ABB RobotStudio station: Práctica5_inicio.rspag

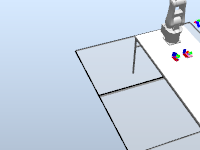
--- station ---
Station Práctica3_inicio (saved by RobotStudio 20.1.9056.2)
Controller Controlador2, task T_ROB1: task frame (RAPID world) sits at (0, 0, 670) mm in the station
Controller Controlador2
  mechanical unit ROB_1: IRB120_3_58__01, 6 joints, base frame (0, 0, 0) mm
Layout (positions relative to the parent item):
  - TVentosa [mechanism] at (-70, 0, 1604) mm
      TCP TVentosa at (0, 0, 51.19) mm
      links: Mi_herramienta
  - LogicGate [smart component, from Components\LogicGate.rslib]
      properties: Operator=NOT; Delay=0
  - LogicGate_2 [smart component, from Components\LogicGate.rslib]
      properties: Operator=AND; Delay=0
  - IRB120_3_58__01 [mechanism, from Robots\IRB120_3_58_G_01.rslib] at (0, 0, 670) mm; joint values [0, 0, -1.5708, 0, 0, 0] (rad or m)
  - table [part, from Libraries\e293a11e-ed86-4237-866f-a9bf8f4bd145table.rslib] at (-246.62, 300, 670) mm, rotated rx 0 ry 0 rz -90 deg
  - Base2 [part]
  - Base1 [part]
  - Detacher [smart component, from Components\Detacher.rslib]
      properties: Child=(none); KeepPosition=true
  - CollisionSensor [smart component, from Components\CollisionSensor.rslib]
      properties: Object1=TVentosa; Object2=(none); NearMiss=0.001; Part1=(none); Part2=(none); CollisionType=0
  - Attacher_2 [smart component, from Components\Attacher.rslib]
      properties: Parent=TVentosa; Flange=0; Child=(none); Mount=false; Offset=[0 0 0]; Orientation=[0 0 0]
  - Source_2 [smart component, from Components\Source.rslib]
      properties: Source=Pieza; Copy=(none); Parent=(none); Position=[0.34 -0.13 0.68]; Orientation=[0 0 0]; Transient=true; PhysicsBehavior=0
  - SimulationEvents_2 [smart component, from Components\SimulationEvents.rslib]
  - Pieza [part] at (340, -130, 700) mm, rotated rx 180 ry 0 rz 180 deg
Attachment: TVentosa is attached to IRB120_3_58__01 / Link6
Attachment: Base2 is attached to Base1
Attachment: Base1 is attached to table
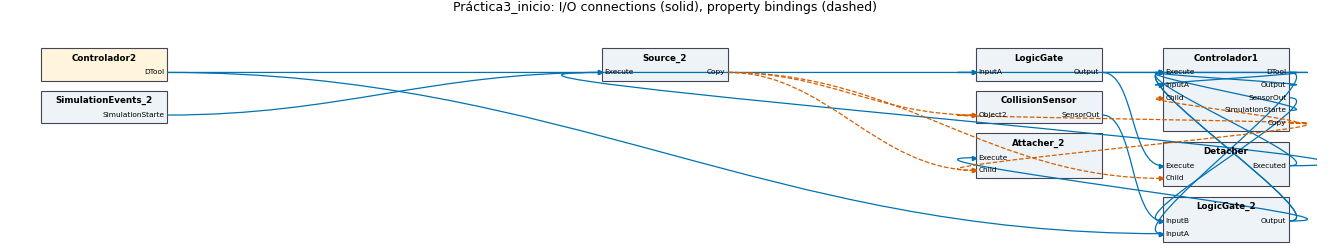
Station logic (signal -> signal, property => property):
  Controlador1.DTool -> Attacher.Execute
  Controlador1.DTool -> LogicGate_2.InputA
  LogicGate_2.Output -> Detacher.Execute
  Controlador1.DTool -> LogicGate.InputA
  LogicGate.Output -> Detacher.Execute
  CollisionSensor.SensorOut -> LogicGate_2.InputB
  Controlador1.DTool -> LogicGate_2.InputA
  LogicGate_2.Output -> Attacher.Execute
  Controlador2.DTool -> LogicGate.InputA
  LogicGate.Output -> Detacher.Execute
  Controlador2.DTool -> LogicGate_2.InputA
  LogicGate_2.Output -> Attacher.Execute
  Detacher.Executed -> Source.Execute
  SimulationEvents.SimulationStarted -> Source.Execute
  CollisionSensor.SensorOut -> LogicGate_2.InputB
  SimulationEvents_2.SimulationStarted -> Source_2.Execute
  Detacher.Executed -> Source_2.Execute
  LogicGate_2.Output -> Attacher_2.Execute
  Source.Copy => Attacher.Child
  Source.Copy => CollisionSensor.Object2
  Source.Copy => Attacher_2.Child
  Source_2.Copy => Attacher_2.Child
  Source_2.Copy => CollisionSensor.Object2
  Source_2.Copy => Detacher.Child

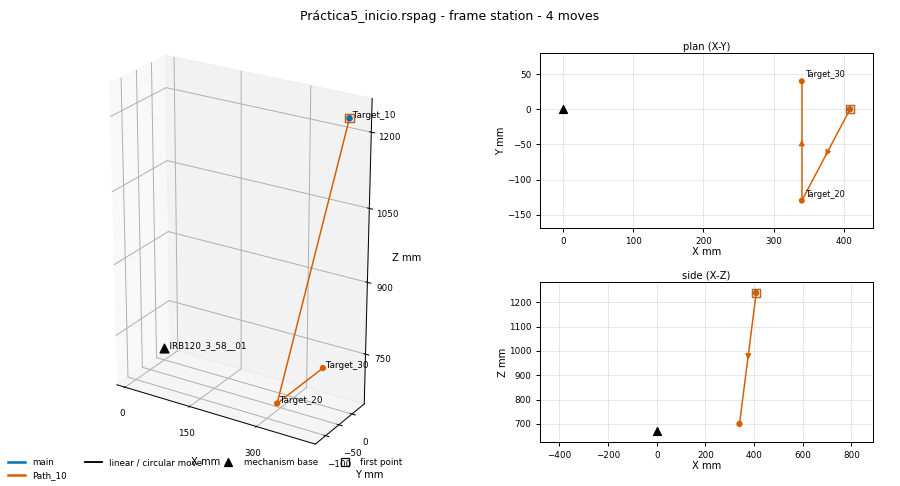
[picture p0: tool path of Práctica5_inicio.rspag in frame station, 4 of 12 moves have a stored position in this frame; points joined in program order, loops and branches not executed]
--- Backups/Controlador2/RAPID/TASK1/PROGMOD/CalibData.mod ---
MODULE CalibData
    PERS tooldata TVentosa:=[TRUE,[[0,0,51.19],[1,0,0,0]],[0.1,[0,0,1],[1,0,0,0],0,0,0]];
    TASK PERS wobjdata WO_Pieza:=[FALSE,TRUE,"",[[300,-150,10],[1,0,0,0]],[[20,10,0],[1,0,0,0]]];
    TASK PERS wobjdata WO_Base2:=[FALSE,TRUE,"",[[300,-150,10],[1,0,0,0]],[[0,150,0],[1,0,0,0]]];
ENDMODULE

--- Backups/Controlador2/RAPID/TASK1/PROGMOD/Module1.mod ---
MODULE Module1
    CONST robtarget Target_10:=[[408.685,0,568.405],[0.5,0,0.866025404,0],[0,0,0,0],[9E+09,9E+09,9E+09,9E+09,9E+09,9E+09]];
    CONST robtarget Target_20:=[[19.999989664,10.000006428,19.999948885],[-0.000000013,0,1,0.000000005],[-1,0,-1,0],[9E+09,9E+09,9E+09,9E+09,9E+09,9E+09]];
    CONST robtarget Target_30:=[[40,40,20],[0,0,1,0],[0,0,0,0],[9E+09,9E+09,9E+09,9E+09,9E+09,9E+09]];
    VAR num h;
    CONST jointtarget JHome:=[[0,0,-90,0,0,0],[9E+09,9E+09,9E+09,9E+09,9E+09,9E+09]];
    !***********************************************************
    !
    ! Módulo:  Module1
    !
    ! Descripción:
    !   <Introduzca la descripción aquí>
    !
    ! Autor: Javier
    !
    ! Versión: 1.0
    !
    !***********************************************************

    PROC main()
        !Añada aquí su código
        Initialize;
        MoveJ Target_10,v200,z100,TVentosa\WObj:=wobj0;
        WHILE DFin = 0 DO
            IF DPieza = 1 THEN
               Pick(Target_20);
               Place(Offs(Target_30,0,0,h));
               h := h + 20;
            ENDIF
        ENDWHILE
        MoveAbsJ JHome,v150,z200,TVentosa\WObj:=WO_Pieza;

    ENDPROC
    PROC Initialize()
        h := 0;
    ENDPROC

    PROC Pick(robtarget posicion)
        MoveL Offs(posicion,0,0,50),v500,z100,TVentosa\WObj:=WO_Pieza;
        MoveL posicion,v200,fine,TVentosa\WObj:=WO_Pieza;
        SetDO DTool,1;
        MoveL Offs(posicion,0,0,50),v200,z100,TVentosa\WObj:=WO_Pieza;
    ENDPROC
    PROC Place(robtarget posicion)
        MoveL Offs(posicion,0,0,50),v500,fine,TVentosa\WObj:=WO_Base2;
        MoveL posicion,v200,fine,TVentosa\WObj:=WO_Base2;
        SetDO DTool,0;
        MoveL Offs(posicion,0,0,50),v200,fine,TVentosa\WObj:=WO_Base2;
    ENDPROC
    PROC Path_10()
        MoveJ Target_10,v200,z100,TVentosa\WObj:=wobj0;
        MoveL Target_20,v200,fine,TVentosa\WObj:=WO_Pieza;
        MoveL Target_30,v200,z100,TVentosa\WObj:=WO_Base2;
        MoveAbsJ JHome,v200,z100,TVentosa\WObj:=WO_Pieza;
    ENDPROC

ENDMODULE

--- Backups/Controlador2/SYSPAR/EIO.cfg ---
EIO:CFG_1.0:6:1::
#
EIO_SIGNAL:

      -Name "DFin" -SignalType "DI"

      -Name "DTool" -SignalType "DO"

      -Name "DPieza" -SignalType "DI"
